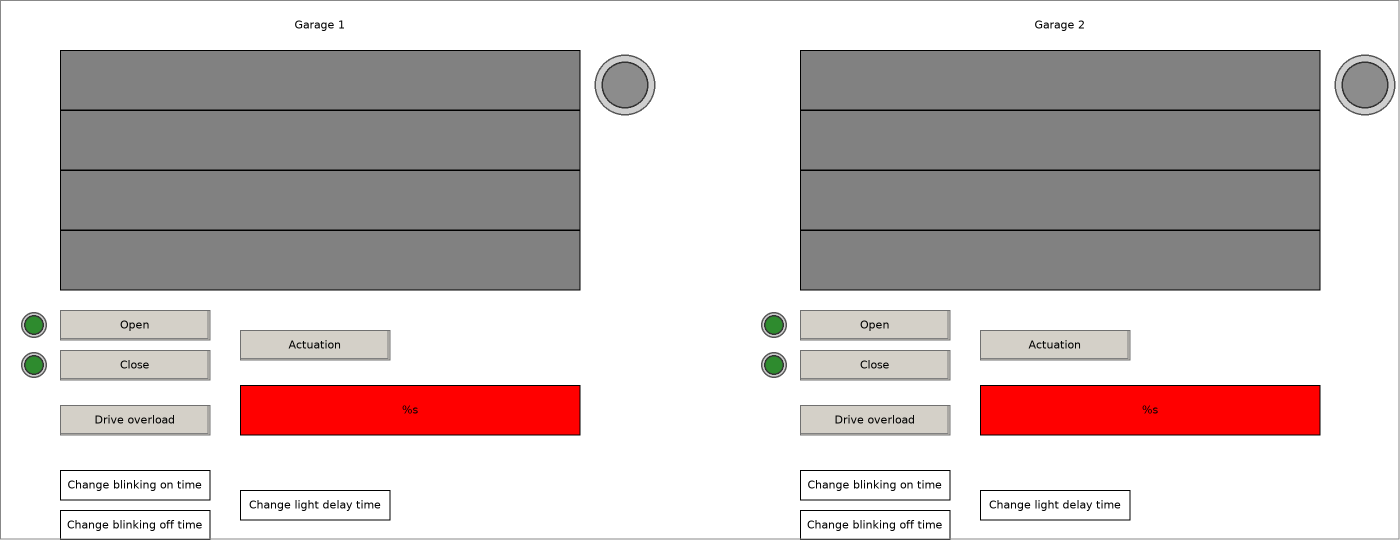
VISUALIZATION Visualization  // 1400x540
    Rectangle (60,50 520x240)
    Rectangle (60,50 520x60), invisible if: MAIN.fbGarage1.Rect2
    Button (240,330 150x30), "Actuation"
        tap MAIN.bActuation1
    Button (60,310 150x30), "Open"
        tap MAIN.bOpenButton1
    Button (60,350 150x30), "Close"
        tap MAIN.bCloseButton1
    Lamp1 (590,50 70x70), variable: MAIN.bDoorLight1, style: Lamp-Lamp1-Gray
    Lamp1 (19,310 30x30), variable: MAIN.bOpeningLight1, style: Lamp-Lamp1-Green
    Lamp1 (19,350 30x30), variable: MAIN.bClosingLight1, style: Lamp-Lamp1-Green
    Rectangle (60,110 520x60), invisible if: MAIN.fbGarage1.Rect2
    Rectangle (60,170 520x60), invisible if: MAIN.fbGarage1.Rect1
    Rectangle (60,230 520x60), invisible if: MAIN.fbGarage1.Rect1
    Button (60,405 150x30), "Drive overload"
        tap MAIN.bDriveOverload1
    Rectangle (800,50 520x240)
    Rectangle (800,50 520x60), invisible if: MAIN.fbGarage2.Rect2
    Button (980,330 150x30), "Actuation"
        tap MAIN.bActuation2
    Button (800,310 150x30), "Open"
        tap MAIN.bOpenButton2
    Button (800,350 150x30), "Close"
        tap MAIN.bCloseButton2
    Lamp1 (1330,50 70x70), variable: MAIN.bDoorLight2, style: Lamp-Lamp1-Gray
    Lamp1 (759,310 30x30), variable: MAIN.bOpeningLight2, style: Lamp-Lamp1-Green
    Lamp1 (759,350 30x30), variable: MAIN.bClosingLight2, style: Lamp-Lamp1-Green
    Rectangle (800,110 520x60), invisible if: MAIN.fbGarage2.Rect2
    Rectangle (800,170 520x60), invisible if: MAIN.fbGarage2.Rect1
    Rectangle (800,230 520x60), invisible if: MAIN.fbGarage2.Rect1
    Button (800,405 150x30), "Drive overload"
        tap MAIN.bDriveOverload2
    Label (245,10 150x30), "Garage 1"
    Label (985,10 150x30), "Garage 2"
    Rectangle (240,385 340x50), "%s", text variable: MAIN.sErrorMessage1, invisible if: MAIN.bNoError1
    Rectangle (980,385 340x50), "%s", text variable: MAIN.sErrorMessage2, invisible if: MAIN.bNoError2
    Rectangle (240,490 150x30), "Change light delay time"
        OnMouseClick: write MAIN.dwLightDelay1 via Default
    Rectangle (60,470 150x30), "Change blinking on time"
        OnMouseClick: write MAIN.dwBlinkingTimeOn1 via Default
    Rectangle (60,510 150x30), "Change blinking off time"
        OnMouseClick: write MAIN.dwBlinkingTimeOff1 via Default
    Rectangle (800,470 150x30), "Change blinking on time"
        OnMouseClick: write MAIN.dwBlinkingTimeOn2 via Default
    Rectangle (800,510 150x30), "Change blinking off time"
        OnMouseClick: write MAIN.dwBlinkingTimeOff2 via Default
    Rectangle (980,490 150x30), "Change light delay time"
        OnMouseClick: write MAIN.dwLightDelay2 via Default
END_VISUALIZATION

(* stored: Version 1.1.0.1, ProductVersion 3.1.4024.12
   Visu Visualization: Id {17d39dcb-2bc6-4375-9880-9249bb2aafad} *)
